PROGRAM P_RunClock_1
VAR
	
	fbClock : FB_Clock;
	
END_VAR


fbClock(
	bStartEnable := G_Enables.bTest,
	fTimeStep := G_Parameters.fTimeStep,
	
	fTime => G_OPC.fTime
);

END_PROGRAM

(* stored: Version 1.1.0.1
   POU P_RunClock_1: Id {ea65958a-3692-4875-9866-2fe082de6fa9}, SpecialFunc None *)
